TYPE stObject :
STRUCT
	x : REAL;
	y : REAL;
	width : REAL;
	height : REAL;
END_STRUCT
END_TYPE

(* stored: Version 1.1.0.1, ProductVersion 3.1.4026.8
   DUT stObject: Id {d7027419-c5c7-435b-9964-7e2915938f52} *)
